PROGRAM POU
VAR
END_VAR

// NETWORK 1

END_PROGRAM

(* stored: Version 1.1.0.1, ProductVersion 3.1.4020.12
   POU POU: Id {8f6c4c87-d845-4b14-863b-5a697965eec8}, SpecialFunc None *)
